// TIA Portal V16 export
// export: Created 2021-11-12T13:31:03.587846Z, ExportSetting WithDefaults, DisplayName Totally Integrated Automation Portal, DisplayVersion V16 Update 3, DisplayName TIA Portal Version Control Interface, DisplayVersion V16 Update 2, DisplayName TIA Portal Openness, DisplayVersion V16 Update 3, DisplayName SINAMICS Startdrive Advanced, DisplayVersion V16 Update 5, DisplayName SINAMICS Startdrive G130, G150, S120, S150, SINAMICS MV, S210, DisplayVersion V16 Update 5, DisplayName SINAMICS Startdrive G110M, G120, G120C, G120D, G120P, G115D, DisplayVersion V16 Update 5, DisplayName STEP 7 Professional, DisplayVersion V16 Update 3, DisplayName STEP 7 Safety, DisplayVersion V16, DisplayName WinCC UA Professional, DisplayVersion V16 Update 3
FUNCTION_BLOCK "Comm"   // FB3, LAD
{ S7_Optimized_Access := 'TRUE' }
VERSION : 0.1
// Communication between main control system and other suppliers control systems
// stored: AutoNumber true, IsIECCheckEnabled false, IsRetainMemResEnabled false, MemoryReserve 100, SetENOAutomatically false, UDAEnableTagReadback false
BEGIN

REGION Network 1: ********* INPUTS ************
END_REGION

REGION Network 2: KAS1 - > CRS
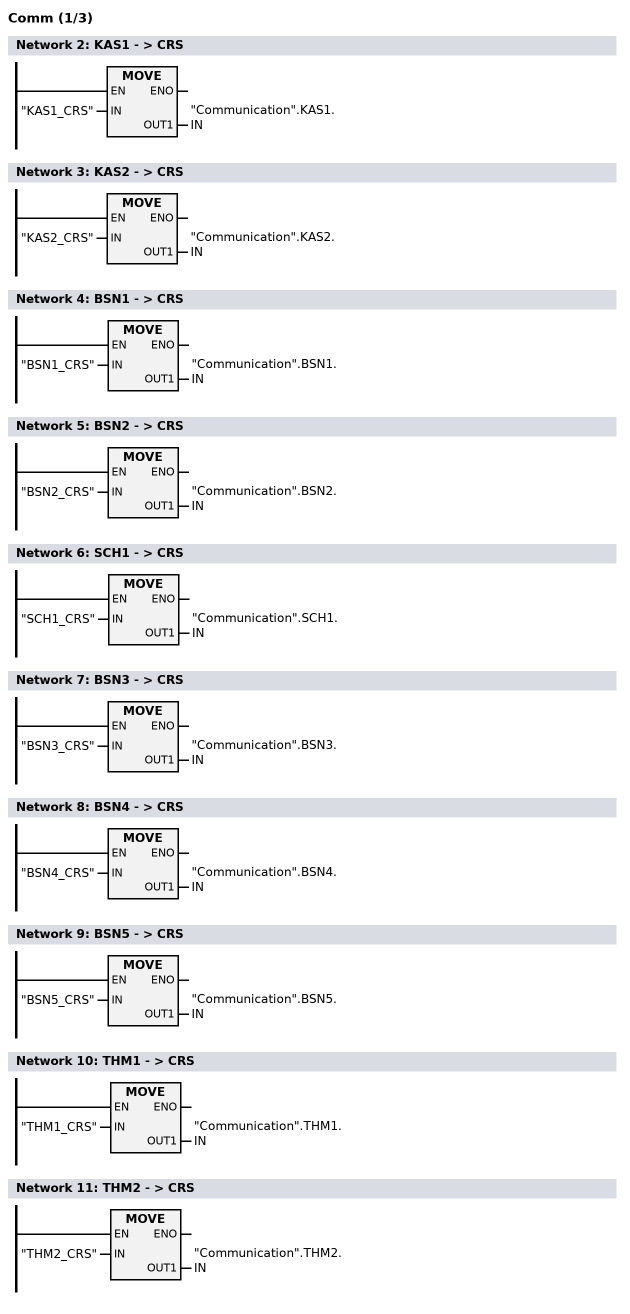
   RUNG wire#powerrail
      Move(in := "KAS1_CRS", out1 => "Communication".KAS1.IN)
   END_RUNG
   // the same network as SCL:
   "Communication".KAS1.IN := "KAS1_CRS";
END_REGION

REGION Network 3: KAS2 - > CRS
   RUNG wire#powerrail
      Move(in := "KAS2_CRS", out1 => "Communication".KAS2.IN)
   END_RUNG
   // the same network as SCL:
   "Communication".KAS2.IN := "KAS2_CRS";
END_REGION

REGION Network 4: BSN1 - > CRS
   RUNG wire#powerrail
      Move(in := "BSN1_CRS", out1 => "Communication".BSN1.IN)
   END_RUNG
   // the same network as SCL:
   "Communication".BSN1.IN := "BSN1_CRS";
END_REGION

REGION Network 5: BSN2 - > CRS
   RUNG wire#powerrail
      Move(in := "BSN2_CRS", out1 => "Communication".BSN2.IN)
   END_RUNG
   // the same network as SCL:
   "Communication".BSN2.IN := "BSN2_CRS";
END_REGION

REGION Network 6: SCH1 - > CRS
   RUNG wire#powerrail
      Move(in := "SCH1_CRS", out1 => "Communication".SCH1.IN)
   END_RUNG
   // the same network as SCL:
   "Communication".SCH1.IN := "SCH1_CRS";
END_REGION

REGION Network 7: BSN3 - > CRS
   RUNG wire#powerrail
      Move(in := "BSN3_CRS", out1 => "Communication".BSN3.IN)
   END_RUNG
   // the same network as SCL:
   "Communication".BSN3.IN := "BSN3_CRS";
END_REGION

REGION Network 8: BSN4 - > CRS
   RUNG wire#powerrail
      Move(in := "BSN4_CRS", out1 => "Communication".BSN4.IN)
   END_RUNG
   // the same network as SCL:
   "Communication".BSN4.IN := "BSN4_CRS";
END_REGION

REGION Network 9: BSN5 - > CRS
   RUNG wire#powerrail
      Move(in := "BSN5_CRS", out1 => "Communication".BSN5.IN)
   END_RUNG
   // the same network as SCL:
   "Communication".BSN5.IN := "BSN5_CRS";
END_REGION

REGION Network 10: THM1 - > CRS
   RUNG wire#powerrail
      Move(in := "THM1_CRS", out1 => "Communication".THM1.IN)
   END_RUNG
   // the same network as SCL:
   "Communication".THM1.IN := "THM1_CRS";
END_REGION

REGION Network 11: THM2 - > CRS
   RUNG wire#powerrail
      Move(in := "THM2_CRS", out1 => "Communication".THM2.IN)
   END_RUNG
   // the same network as SCL:
   "Communication".THM2.IN := "THM2_CRS";
END_REGION

REGION Network 12: MEM1 - > CRS
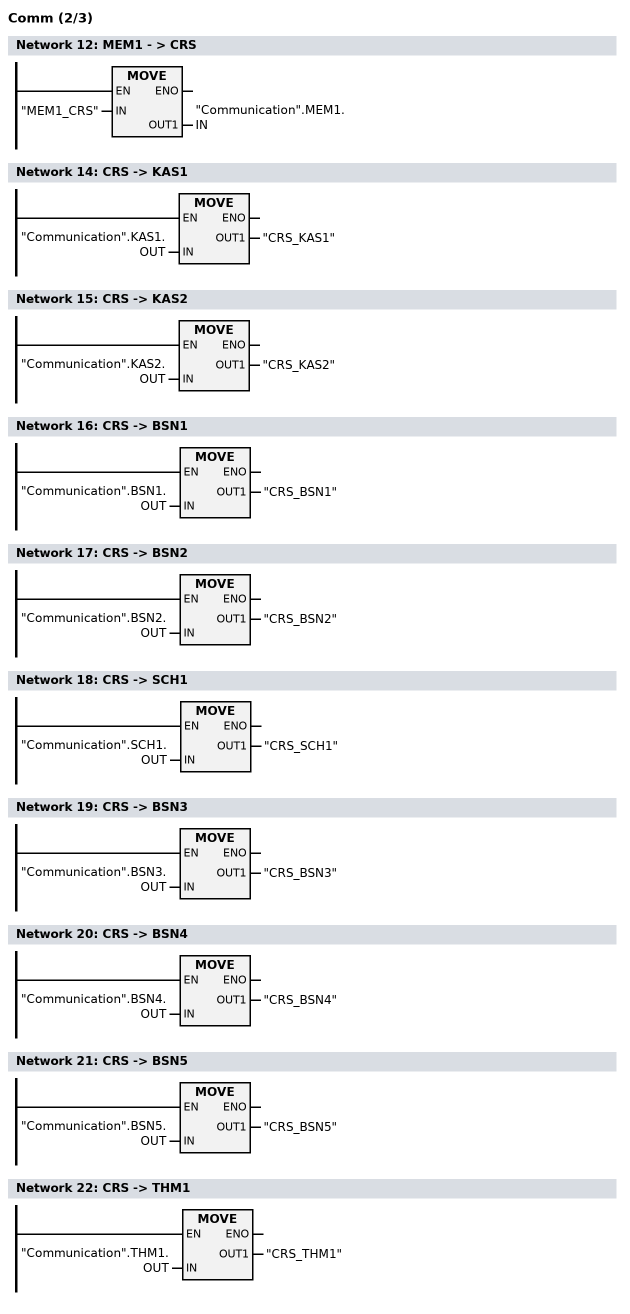
   RUNG wire#powerrail
      Move(in := "MEM1_CRS", out1 => "Communication".MEM1.IN)
   END_RUNG
   // the same network as SCL:
   "Communication".MEM1.IN := "MEM1_CRS";
END_REGION

REGION Network 13: ********* OUTPUTS ************
END_REGION

REGION Network 14: CRS -> KAS1
   RUNG wire#powerrail
      Move(in := "Communication".KAS1.OUT, out1 => "CRS_KAS1")
   END_RUNG
   // the same network as SCL:
   "CRS_KAS1" := "Communication".KAS1.OUT;
END_REGION

REGION Network 15: CRS -> KAS2
   RUNG wire#powerrail
      Move(in := "Communication".KAS2.OUT, out1 => "CRS_KAS2")
   END_RUNG
   // the same network as SCL:
   "CRS_KAS2" := "Communication".KAS2.OUT;
END_REGION

REGION Network 16: CRS -> BSN1
   RUNG wire#powerrail
      Move(in := "Communication".BSN1.OUT, out1 => "CRS_BSN1")
   END_RUNG
   // the same network as SCL:
   "CRS_BSN1" := "Communication".BSN1.OUT;
END_REGION

REGION Network 17: CRS -> BSN2
   RUNG wire#powerrail
      Move(in := "Communication".BSN2.OUT, out1 => "CRS_BSN2")
   END_RUNG
   // the same network as SCL:
   "CRS_BSN2" := "Communication".BSN2.OUT;
END_REGION

REGION Network 18: CRS -> SCH1
   RUNG wire#powerrail
      Move(in := "Communication".SCH1.OUT, out1 => "CRS_SCH1")
   END_RUNG
   // the same network as SCL:
   "CRS_SCH1" := "Communication".SCH1.OUT;
END_REGION

REGION Network 19: CRS -> BSN3
   RUNG wire#powerrail
      Move(in := "Communication".BSN3.OUT, out1 => "CRS_BSN3")
   END_RUNG
   // the same network as SCL:
   "CRS_BSN3" := "Communication".BSN3.OUT;
END_REGION

REGION Network 20: CRS -> BSN4
   RUNG wire#powerrail
      Move(in := "Communication".BSN4.OUT, out1 => "CRS_BSN4")
   END_RUNG
   // the same network as SCL:
   "CRS_BSN4" := "Communication".BSN4.OUT;
END_REGION

REGION Network 21: CRS -> BSN5
   RUNG wire#powerrail
      Move(in := "Communication".BSN5.OUT, out1 => "CRS_BSN5")
   END_RUNG
   // the same network as SCL:
   "CRS_BSN5" := "Communication".BSN5.OUT;
END_REGION

REGION Network 22: CRS -> THM1
   RUNG wire#powerrail
      Move(in := "Communication".THM1.OUT, out1 => "CRS_THM1")
   END_RUNG
   // the same network as SCL:
   "CRS_THM1" := "Communication".THM1.OUT;
END_REGION

REGION Network 23: CRS -> THM2
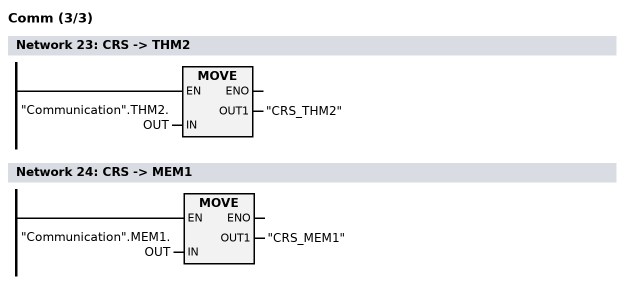
   RUNG wire#powerrail
      Move(in := "Communication".THM2.OUT, out1 => "CRS_THM2")
   END_RUNG
   // the same network as SCL:
   "CRS_THM2" := "Communication".THM2.OUT;
END_REGION

REGION Network 24: CRS -> MEM1
   RUNG wire#powerrail
      Move(in := "Communication".MEM1.OUT, out1 => "CRS_MEM1")
   END_RUNG
   // the same network as SCL:
   "CRS_MEM1" := "Communication".MEM1.OUT;
END_REGION
END_FUNCTION_BLOCK
